// TIA Portal project "Insert_Password" (V18)

(* hardware
DEVICE "S7-1200 station_2"  S7-1200 Station
   slot 0: "Rack_0"  S7-1200 Rack  Rack  V1.0
   slot 1: "PLC_1"  CPU 1215C DC/DC/Rly  6ES7 215-1HG40-0XB0  V4.6
DEVICE "HMI_1"  KTP700 Basic PN
   slot 0: "HMI_1"  KTP700 Basic PN  6AV2 123-2GB03-0AX0  17.0.0.0
   slot 1: "HMI_RT_1"  KTP700 Basic PN  6AV2 123-2GB03-0AX0  17.0.0.0
   slot 5: "HMI_1.IE_CP_1"  PROFINET Interface  17.0.0.0
      slot 1: "PROFINET Interface_1"  PROFINET Interface
         slot 1: "Port_1"  Port
*)

// ===== PLC "PLC_1"  CPU 1215C DC/DC/Rly =====

VAR_GLOBAL   // PLC tag table "Default tag table"
   "Clock_Byte" AT %MB0 : Byte;
   "Clock_10Hz" AT %M0.0 : Bool;
   "Clock_5Hz" AT %M0.1 : Bool;
   "Clock_2.5Hz" AT %M0.2 : Bool;
   "Clock_2Hz" AT %M0.3 : Bool;
   "Clock_1.25Hz" AT %M0.4 : Bool;
   "Clock_1Hz" AT %M0.5 : Bool;
   "Clock_0.625Hz" AT %M0.6 : Bool;
   "Clock_0.5Hz" AT %M0.7 : Bool;
END_VAR

DATA_BLOCK "Logica_TIP_DB"   // DB1
{ S7_Optimized_Access := 'TRUE' }
VERSION : 0.1
// stored: InstanceOfName Logica_TIP
"Logica_TIP"
BEGIN
END_DATA_BLOCK

DATA_BLOCK "Data_block_1"   // DB3
{ S7_Optimized_Access := 'TRUE' }
VERSION : 0.1
   VAR
      Convalida_Lv1 : Bool;
      Convalida_Lv2 : Bool;
      Convalida_Lv3 : Bool;
      Disattiva : Bool;
      Selezione_modalita : Int;
      Password_1 : Array[0..15] of UInt;
      Password_2 : Array[0..15] of UInt;
      Password_3 : Array[0..15] of UInt;
      Lunghezza_Pw : Int := 8;
      richiesta_lv1 : Bool;
      richiesta_lv2 : Bool;
      richiesta_lv3 : Bool;
   END_VAR
BEGIN
   Password_1[0] := 1;
   Password_1[1] := 2;
   Password_1[2] := 1;
   Password_1[3] := 1;
   Password_2[0] := 0;
   Password_2[1] := 4;
   Password_2[2] := 0;
   Password_2[3] := 9;
   Password_3[0] := 1;
   Password_3[1] := 2;
   Password_3[2] := 3;
   Password_3[3] := 4;
   Password_1[4] := 2;
   Password_1[5] := 0;
   Password_1[6] := 2;
   Password_1[7] := 3;
   Password_2[4] := 1;
   Password_2[5] := 9;
   Password_2[6] := 9;
   Password_2[7] := 7;
   Password_3[4] := 5;
   Password_3[5] := 6;
   Password_3[6] := 7;
   Password_3[7] := 8;
   Password_3[8] := 0;
   Password_3[9] := 0;
END_DATA_BLOCK

// folder: System blocks/Program resources

DATA_BLOCK "IEC_Timer_0_DB"   // DB2
{ S7_Optimized_Access := 'TRUE' }
AUTHOR : Simatic
FAMILY : IEC
NAME : IEC_TMR
VERSION : 1.0
// stored: InstanceOfName IEC_TIMER
"IEC_TIMER"
BEGIN
END_DATA_BLOCK

DATA_BLOCK "IEC_Timer_0_DB_1"   // DB4
{ S7_Optimized_Access := 'TRUE' }
AUTHOR : Simatic
FAMILY : IEC
NAME : IEC_TMR
VERSION : 1.0
// stored: InstanceOfName IEC_TIMER
"IEC_TIMER"
BEGIN
END_DATA_BLOCK

// folder: (top level)

FUNCTION_BLOCK "Logica_TIP"   // FB2, SCL
{ S7_Optimized_Access := 'TRUE' }
VERSION : 0.1
   VAR_INPUT
      Selezione_Modalità : Int;
      Richiesta_Lv_1 : Bool;
      Richiesta_Lv_2 : Bool;
      Richiesta_Lv_3 : Bool;
      Disattiva_Abilitazioni : Bool;
   END_VAR
   VAR_OUTPUT
      Livello_1 : Bool;
      Livello_2 : Bool;
      Livello_3 : Bool;
   END_VAR
   VAR_IN_OUT
      password_1 : Array[0..#N_Array] of UInt;
      password_2 : Array[0..#N_Array] of UInt;
      password_3 : Array[0..#N_Array] of UInt;
      Lunghezza_Pw : Int;
   END_VAR
   VAR
      Array_Input : Array[0..#N_Array] of UInt;
      Array_Linee : Array[0..#N_Array] of Bool;
      Conteggio : UInt;
      Array_Memoria : Array[0..#N_Array] of Bool;
      Array_Fronti : Array[0..#N_Array] of Bool;
      Array_Fronti_Change : Array[0..#N_Array] of Bool;
      Visibilità : Bool;
      Numero : UInt;
      visibilità_Numeri : UInt;
      "Visibilità_Numeri_*" : UInt;
      "Visibilità_Numeri_°" : UInt;
      Attiva_Change : Bool;
      Stato_Cambio_Pw : UInt;
      Richiesta_Lv1 : Bool;
      Richiesta_Lv2 : Bool;
      Richiesta_Lv3 : Bool;
      Fronte_Disabilità : Bool;
      Variabili_Scritte_Change : String;
      Change_Status : UInt;
      "Password_Selected_ Change" : UInt;
      ET : Time;
      ET_1 : Time;
      appoggio_fronte_10 : Bool;
      n_div : Array[0..10] of Int;
      Scritte_Errori : String;
      vis_Scritte_Errori : Bool;
      R1 : R_TRIG;
      R2 : R_TRIG;
      R3 : R_TRIG;
      R4 : R_TRIG;
      R5 : R_TRIG;
      F_13 : F_TRIG;
      R_11 : R_TRIG;
      R_12 : R_TRIG;
      R_14 : R_TRIG;
      R_0 : R_TRIG;
      R_1 : R_TRIG;
      R_3 : R_TRIG;
      R_4 : R_TRIG;
      R_5 : R_TRIG;
      R_6 : R_TRIG;
      R_2 : R_TRIG;
      R_7 : R_TRIG;
      R_8 : R_TRIG;
      R_9 : R_TRIG;
   END_VAR
   VAR_TEMP
      n : Int;
   END_VAR
   VAR CONSTANT
      N_Array : Int := 15;
   END_VAR
BEGIN
   IF #Lunghezza_Pw > 16 THEN
       #Lunghezza_Pw := 16;
       #Scritte_Errori := 'Valore massimo inseribile: 16';
       #vis_Scritte_Errori := true;
   END_IF;

   REGION monitoro le richieste abilitazioni e attivo i vari settaggi
       #R1(CLK:=#Richiesta_Lv_1);
       #R2(CLK:=#Richiesta_Lv_2);
       #R3(CLK:=#Richiesta_Lv_3);

       IF #R1.Q THEN
           #Visibilità := true;
           #Richiesta_Lv1 := true;
       END_IF;

       IF #R2.Q THEN
           #Visibilità := true;
           #Richiesta_Lv2 := true;
       END_IF;

       IF #R3.Q THEN
           #Visibilità := true;
           #Richiesta_Lv3 := true;
       END_IF;
   END_REGION

   REGION Gestione attivazione Visibilità
       #R4(CLK := #Visibilità);
       IF #R4.Q THEN
           #Variabili_Scritte_Change := 'inserisci password';
           #visibilità_Numeri := 1;
           #Conteggio := 0;
       END_IF;
   END_REGION;

   IF #Visibilità = TRUE THEN  //verifico se la visibilità è attiva
       REGION gestione linee e numeri/asterischi
           IF "Clock_1.25Hz" = true THEN
               #Array_Linee[#Conteggio] := true;
           ELSE
               FOR #n := 0 TO #N_Array DO
                   #Array_Linee[#n] := FALSE;
               END_FOR;
           END_IF;

           #R5(CLK:="Clock_10Hz");
           IF #R5.Q THEN
               FOR #n := 0 TO #N_Array DO
                   #Array_Linee[#n] := FALSE;
               END_FOR;
           END_IF;

           #F_13(CLK:=#Array_Memoria[13]);

           IF #Array_Memoria[13] = true THEN
               #visibilità_Numeri := 2;
           END_IF;

           IF #F_13.Q THEN
               IF "IEC_Timer_0_DB_1".Q = true THEN
                   #visibilità_Numeri := 2;
               ELSE
                   #visibilità_Numeri := 1;
               END_IF;
           END_IF;


           "IEC_Timer_0_DB_1".TON(IN := #Array_Memoria[13],
                                  PT := T#1s,
                                  ET => #ET);

           CASE #visibilità_Numeri OF
               1:
                   #"Visibilità_Numeri_°" := 0;
                   #"Visibilità_Numeri_*" := #Lunghezza_Pw;
               2:
                   #"Visibilità_Numeri_°" := #Lunghezza_Pw;
                   #"Visibilità_Numeri_*" := 0;

           END_CASE;
       END_REGION

       REGION rilevamento e gestione pulsanti 
           REGION rilevamento e funzionalita pulsante esc
               // pressione pulsante "ESC"
               #R_11(CLK:=#Array_Memoria[11]);

               IF #R_11.Q THEN
                   FOR #n := 0 TO #N_Array DO
                       #Array_Input[#n] := 0;
                   END_FOR;
                   FOR #n := 0 TO #N_Array DO
                       #Array_Linee[#n] := FALSE;
                   END_FOR;
                   #Conteggio := 0;
                   #Visibilità := FALSE;
                   #Richiesta_Lv1 := false;
                   #Richiesta_Lv2 := false;
                   #Richiesta_Lv3 := false;
                   #"Visibilità_Numeri_°" := 0;
                   #"Visibilità_Numeri_*" := 0;
                   #Change_Status := 0;
               END_IF;
           END_REGION

           REGION rilevamento e funzionalità pulsante canc
               // pressione pulsante "CANC"
               #R_12(CLK:=#Array_Memoria[12]);
               IF #R_12.Q THEN
                   FOR #n := 0 TO #N_Array DO
                       #Array_Input[#n] := 0;
                   END_FOR;
                   #Conteggio := 0;
               END_IF;
           END_REGION

           REGION rilevamento e funzionalità pulsante indietro
               // pressione pulsante indietro
               #R_14(CLK:=#Array_Memoria[14]);
               IF #R_14.Q THEN
                   IF #Conteggio > 0 THEN
                       #Conteggio := #Conteggio - 1;
                       #Array_Input[#Conteggio] := 0;
                   END_IF;
               END_IF;
           END_REGION

       END_REGION

       REGION rilevazione pressione pulsanti fintanto che il numero di caratteri inseriti non superi la lunghezza_pw

           IF #Conteggio < #Lunghezza_Pw THEN  //verifico se le volte in cui i numeri sono stati premuti è minore di #lunghezza_pw

               //vado a registrare gli input dei pulsanti numerici
               #R_0(CLK:= #Array_Memoria[0]);
               #R_1(CLK:= #Array_Memoria[1]);
               #R_2(CLK:= #Array_Memoria[2]);
               #R_3(CLK:= #Array_Memoria[3]);
               #R_4(CLK := #Array_Memoria[4]);
               #R_5(CLK:= #Array_Memoria[5]);
               #R_6(CLK:= #Array_Memoria[6]);
               #R_7(CLK:= #Array_Memoria[7]);
               #R_8(CLK:= #Array_Memoria[8]);
               #R_9(CLK:= #Array_Memoria[9]);

               IF #R_0.Q THEN
                   #Array_Linee[#Numero] := FALSE;
                   #Array_Input[#Conteggio] := 0;
                   #Conteggio := #Conteggio + 1;
               END_IF;

               IF #R_1.Q THEN
                   #Array_Linee[#Numero] := FALSE;
                   #Array_Input[#Conteggio] := 1;
                   #Conteggio := #Conteggio + 1;
               END_IF;

               IF #R_2.Q  THEN
                   #Array_Linee[#Numero] := FALSE;
                   #Array_Input[#Conteggio] := 2;
                   #Conteggio := #Conteggio + 1;
               END_IF;

               IF #R_3.Q THEN
                   #Array_Linee[#Numero] := FALSE;
                   #Array_Input[#Conteggio] := 3;
                   #Conteggio := #Conteggio + 1;
               END_IF;

               IF #R_4.Q THEN
                   #Array_Linee[#Numero] := FALSE;
                   #Array_Input[#Conteggio] := 4;
                   #Conteggio := #Conteggio + 1;
               END_IF;

               IF #R_5.Q THEN
                   #Array_Linee[#Numero] := FALSE;
                   #Array_Input[#Conteggio] := 5;
                   #Conteggio := #Conteggio + 1;
               END_IF;

               IF #R_6.Q THEN
                   #Array_Linee[#Numero] := FALSE;
                   #Array_Input[#Conteggio] := 6;
                   #Conteggio := #Conteggio + 1;
               END_IF;

               IF #R_7.Q THEN
                   #Array_Linee[#Numero] := FALSE;
                   #Array_Input[#Conteggio] := 7;
                   #Conteggio := #Conteggio + 1;
               END_IF;

               IF #R_8.Q THEN
                   #Array_Linee[#Numero] := FALSE;
                   #Array_Input[#Conteggio] := 8;
                   #Conteggio := #Conteggio + 1;
               END_IF;

               IF #R_9.Q THEN
                   #Array_Linee[#Numero] := FALSE;
                   #Array_Input[#Conteggio] := 9;
                   #Conteggio := #Conteggio + 1;
               END_IF;

           END_IF;
       END_REGION

       REGION Change_Status=0
           IF #Change_Status = 0 THEN

               REGION Restituzione risultato in base alla MODalità di funzionamento selezionata

                   IF (#Array_Memoria[10] = true) & (#Array_Fronti[10] = false) THEN

                       CASE #Selezione_Modalità OF
                           0:
                               FOR #n := 0 TO (#Lunghezza_Pw - 1) DO
                                   IF #Array_Input[#n] <> #password_1[#n] THEN
                                       #n_div[0] := #n_div[0] + 1;
                                   END_IF;
                               END_FOR;
                               FOR #n := 0 TO (#Lunghezza_Pw - 1) DO
                                   IF #Array_Input[#n] <> #password_2[#n] THEN
                                       #n_div[1] := #n_div[1] + 1;
                                   END_IF;
                               END_FOR;
                               FOR #n := 0 TO (#Lunghezza_Pw - 1) DO
                                   IF #Array_Input[#n] <> #password_3[#n] THEN
                                       #n_div[2] := #n_div[2] + 1;
                                   END_IF;
                               END_FOR;
                               IF #n_div[0] = 0 THEN
                                   #Livello_1 := true;
                                   #Livello_2 := true;
                                   #Livello_3 := true;
                                   #Variabili_Scritte_Change := 'Password corretta';
                               ELSE
                                   IF #n_div[1] = 0 THEN
                                       #Livello_2 := true;
                                       #Livello_3 := true;
                                       #Variabili_Scritte_Change := 'Password corretta';
                                   ELSE
                                       IF #n_div[2] = 0 THEN
                                           #Livello_3 := true;
                                           #Variabili_Scritte_Change := 'Password corretta';
                                       ELSE
                                           #Variabili_Scritte_Change := 'Password sbagliata';
                                       END_IF;
                                   END_IF;
                               END_IF;

                                   1:
                                   IF #Richiesta_Lv1 = true THEN
                                       FOR #n := 0 TO (#Lunghezza_Pw - 1) DO
                                           IF #Array_Input[#n] <> #password_1[#n] THEN
                                               #n_div[3] := #n_div[3] + 1;
                                           END_IF;
                                       END_FOR;
                                       IF #n_div[3] = 0 THEN
                                           #Variabili_Scritte_Change := 'Password corretta';
                                           #Livello_1 := true;
                                       ELSE
                                           #Variabili_Scritte_Change := 'Password sbagliata';
                                       END_IF;
                                   END_IF;

                                   IF #Richiesta_Lv2 = true THEN
                                       FOR #n := 0 TO (#Lunghezza_Pw - 1) DO
                                           IF #Array_Input[#n] <> #password_2[#n] THEN
                                               #n_div[4] := #n_div[4] + 1;
                                           END_IF;
                                       END_FOR;
                                       IF #n_div[4] = 0 THEN
                                           #Variabili_Scritte_Change := 'Password corretta';
                                           #Livello_2 := true;
                                       ELSE
                                           #Variabili_Scritte_Change := 'Password sbagliata';
                                       END_IF;
                                   END_IF;

                                   IF #Richiesta_Lv3 = true THEN
                                       FOR #n := 0 TO (#Lunghezza_Pw - 1) DO
                                           IF #Array_Input[#n] <> #password_3[#n] THEN
                                               #n_div[5] := #n_div[5] + 1;
                                           END_IF;
                                       END_FOR;
                                       IF #n_div[5] = 0 THEN
                                           #Variabili_Scritte_Change := 'Password corretta';
                                           #Livello_3 := true;
                                       ELSE
                                           #Variabili_Scritte_Change := 'Password sbagliata';
                                       END_IF;
                                   END_IF;
                                   2:

                                   FOR #n := 0 TO (#Lunghezza_Pw - 1) DO
                                       IF #Array_Input[#n] <> #password_1[#n] THEN
                                           #n_div[6] := #n_div[6] + 1;
                                       END_IF;
                                   END_FOR;
                                   IF #n_div[6] = 0 THEN
                                       #Variabili_Scritte_Change := 'Password corretta';
                                       #Livello_1 := true;
                                       #Livello_2 := true;
                                       #Livello_3 := true;
                                   ELSE
                                       #Variabili_Scritte_Change := 'Password sbagliata';
                                   END_IF;
                       END_CASE;
                   END_IF;
                   #Array_Fronti[10] := #Array_Memoria[10];
                   #Array_Memoria[10] := false;
                   FOR #n := 0 TO 6 DO
                       #n_div[#n] := 0;
                   END_FOR;

               END_REGION

           END_IF;

       END_REGION

       REGION gestione modalità cambio password

           REGION Pressione pulsante change password ed entrata nella modalità sovrascrittura
               IF (#Array_Memoria[15] = true) & (#Array_Fronti[15] = false) THEN
                   #Variabili_Scritte_Change := 'Seleziona password';
                   FOR #n := 0 TO #N_Array DO
                       #Array_Input[#n] := 0;
                   END_FOR;
                   #Conteggio := 0;
                   #Change_Status := 1;
               END_IF;
               #Array_Fronti[15] := #Array_Memoria[15];
           END_REGION

           REGION Change_Status=1

               IF #Change_Status = 1 THEN
                   IF (#Array_Memoria[1] = true) & (#Array_Fronti_Change[1] = false) THEN
                       FOR #n := 0 TO #N_Array DO
                           #Array_Input[#n] := 0;
                       END_FOR;
                       #Conteggio := 0;
                       #Variabili_Scritte_Change := 'password precedente';
                       #Change_Status := 2;
                       #"Password_Selected_ Change" := 1;
                   END_IF;
                   #Array_Fronti_Change[1] := #Array_Memoria[1];

                   IF (#Array_Memoria[2] = true) & (#Array_Fronti_Change[2] = false) THEN
                       FOR #n := 0 TO #N_Array DO
                           #Array_Input[#n] := 0;
                       END_FOR;
                       #Conteggio := 0;
                       #Variabili_Scritte_Change := 'password precedente'; // 
                       #Change_Status := 2;
                       #"Password_Selected_ Change" := 2;
                   END_IF;
                   #Array_Fronti_Change[2] := #Array_Memoria[2];


                   IF (#Array_Memoria[3] = true) & (#Array_Fronti_Change[3] = false) THEN
                       FOR #n := 0 TO #N_Array DO
                           #Array_Input[#n] := 0;
                       END_FOR;
                       #Conteggio := 0;
                       #Variabili_Scritte_Change := 'password precedente';
                       #Change_Status := 2;
                       #"Password_Selected_ Change" := 3;
                   END_IF;
                   #Array_Fronti_Change[3] := #Array_Memoria[3];
               END_IF;

           END_REGION


           REGION Change_Status=2
               IF #Change_Status = 2 THEN
                   IF #Array_Memoria[10] = true & #Array_Fronti_Change[10] = FALSE THEN
                       CASE #"Password_Selected_ Change" OF
                           1:
                               FOR #n := 0 TO (#Lunghezza_Pw - 1) DO
                                   IF #Array_Input[#n] <> #password_1[#n] THEN
                                       #n_div[7] := #n_div[7] + 1;
                                   END_IF;
                               END_FOR;
                               IF #n_div[7] = 0  THEN
                                   #Change_Status := 3;
                                   FOR #n := 0 TO #N_Array DO
                                       #Array_Input[#n] := 0;
                                   END_FOR;
                                   #Conteggio := 0;
                                   #Variabili_Scritte_Change := 'Nuova password';
                                   GOTO end;
                               ELSE
                                   #Variabili_Scritte_Change := 'Password errata';
                               END_IF;

                           2:
                               FOR #n := 0 TO (#Lunghezza_Pw - 1) DO
                                   IF #Array_Input[#n] <> #password_2[#n] THEN
                                       #n_div[8] := #n_div[8] + 1;
                                   END_IF;
                               END_FOR;
                               IF #n_div[8] = 0 THEN
                                   #Change_Status := 3;
                                   FOR #n := 0 TO #N_Array DO
                                       #Array_Input[#n] := 0;
                                   END_FOR;
                                   #Conteggio := 0;
                                   #Variabili_Scritte_Change := 'Nuova password';
                                   GOTO end;
                               ELSE
                                   #Variabili_Scritte_Change := 'Password errata';
                               END_IF;
                           3:
                               FOR #n := 0 TO (#Lunghezza_Pw - 1) DO
                                   IF #Array_Input[#n] <> #password_3[#n] THEN
                                       #n_div[9] := #n_div[9] + 1;
                                   END_IF;
                               END_FOR;
                               IF #n_div[9] = 0 THEN
                                   #Change_Status := 3;
                                   FOR #n := 0 TO #N_Array DO
                                       #Array_Input[#n] := 0;
                                   END_FOR;
                                   #Conteggio := 0;
                                   #Variabili_Scritte_Change := 'Nuova password';
                                   GOTO end;
                               ELSE
                                   #Variabili_Scritte_Change := 'Password errata';
                               END_IF;
                       END_CASE;
                   END_IF;
                   #Array_Fronti_Change[10] := #Array_Memoria[10];
               END_IF;


           END_REGION


           REGION Change_Status=3
               IF #Change_Status = 3 THEN
                   IF #Array_Memoria[10] = true & #Array_Fronti_Change[11] = FALSE THEN
                       #appoggio_fronte_10 := true;
                       #Variabili_Scritte_Change := 'Password modificata';
                   END_IF;
                   "IEC_Timer_0_DB".TON(IN := #appoggio_fronte_10,
                                        PT := T#1s,
                                        ET => #ET_1);
                   IF "IEC_Timer_0_DB".Q = true THEN
                       #appoggio_fronte_10 := false;
                       CASE #"Password_Selected_ Change" OF
                           1:
                               #"password_1" := #Array_Input;
                               GOTO esc;
                           2:
                               #"password_2" := #Array_Input;
                               GOTO esc;
                           3:
                               #"password_3" := #Array_Input;
                               GOTO esc;
                       END_CASE;
                   esc:
                       FOR #n := 0 TO #N_Array DO
                           #Array_Input[#n] := 0;
                       END_FOR;
                       FOR #n := 0 TO #N_Array DO
                           #Array_Linee[#n] := FALSE;
                       END_FOR;
                       #Conteggio := 0;
                       #Visibilità := FALSE;
                       #Richiesta_Lv1 := false;
                       #Richiesta_Lv2 := false;
                       #Richiesta_Lv3 := false;
                       #"Visibilità_Numeri_°" := 0;
                       #"Visibilità_Numeri_*" := 0;
                       #Change_Status := 0;
                   END_IF;
                   #Array_Fronti_Change[11] := #Array_Memoria[10];
                   #Array_Memoria[10] := false;
               END_IF;


           END_REGION

       end:
           #Array_Memoria[10] := false;
           FOR #n := 7 TO 9 DO
               #n_div[#n] := 0;
           END_FOR;
       END_REGION


   END_IF;

   REGION rilevamento e funzionalità pulsante disattiva abilitazioni
       // va fuori dal controllo visibilità altrimenti non funziona
       IF #Disattiva_Abilitazioni = true & #Fronte_Disabilità = false THEN
           #Livello_1 := false;
           #Livello_2 := false;
           #Livello_3 := false;
       END_IF;
       #Fronte_Disabilità := #Disattiva_Abilitazioni;
   END_REGION
END_FUNCTION_BLOCK

ORGANIZATION_BLOCK "Main"   // OB1, LAD, ProgramCycle
TITLE = "Main Program Sweep (Cycle)"
{ S7_Optimized_Access := 'TRUE' }
VERSION : 0.1
   VAR_INPUT
      Initial_Call : Bool;   // Initial call of this OB
      Remanence : Bool;   // =True, if remanent data are available
   END_VAR
BEGIN

REGION Network 1
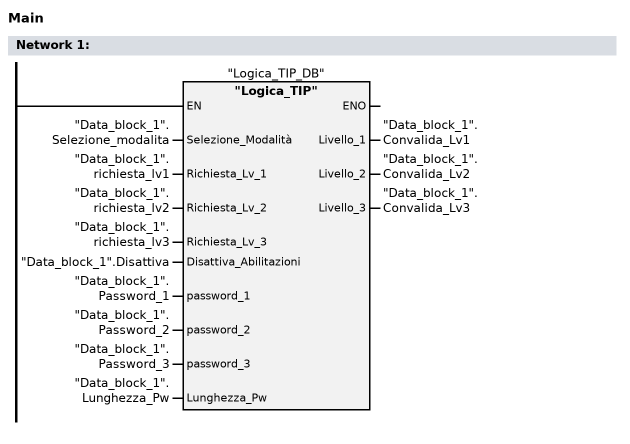
   RUNG wire#powerrail
      "Logica_TIP_DB"(Selezione_Modalità := "Data_block_1".Selezione_modalita, Richiesta_Lv_1 := "Data_block_1".richiesta_lv1, Richiesta_Lv_2 := "Data_block_1".richiesta_lv2, Richiesta_Lv_3 := "Data_block_1".richiesta_lv3, Disattiva_Abilitazioni := "Data_block_1".Disattiva, Lunghezza_Pw := "Data_block_1".Lunghezza_Pw, password_1 := "Data_block_1".Password_1, password_2 := "Data_block_1".Password_2, password_3 := "Data_block_1".Password_3, Livello_1 => "Data_block_1".Convalida_Lv1, Livello_2 => "Data_block_1".Convalida_Lv2, Livello_3 => "Data_block_1".Convalida_Lv3)
   END_RUNG
   // the same network as SCL:
   "Logica_TIP_DB"(Selezione_Modalità := "Data_block_1".Selezione_modalita,   // "Logica_TIP"
                   Richiesta_Lv_1 := "Data_block_1".richiesta_lv1,
                   Richiesta_Lv_2 := "Data_block_1".richiesta_lv2,
                   Richiesta_Lv_3 := "Data_block_1".richiesta_lv3,
                   Disattiva_Abilitazioni := "Data_block_1".Disattiva,
                   password_1 := "Data_block_1".Password_1,
                   password_2 := "Data_block_1".Password_2,
                   password_3 := "Data_block_1".Password_3,
                   Lunghezza_Pw := "Data_block_1".Lunghezza_Pw,
                   Livello_1 => "Data_block_1".Convalida_Lv1,
                   Livello_2 => "Data_block_1".Convalida_Lv2,
                   Livello_3 => "Data_block_1".Convalida_Lv3);
END_REGION
END_ORGANIZATION_BLOCK

(* ===== HMI "HMI_RT_1" =====
system functions are stored by id; their names below are inferred from use
connection "HMI_Connection_1": ETHERNET, SMART_S7_1200_OMS

HMI tags "Default tag table"
   "Tag_ScreenNumber" : UInt, internal
   "Variabili_Visibilità" : Bool = PLC Logica_TIP_DB.Visibilità, 100 ms
   "Variabili_Array_Memoria{12}" : Bool = PLC Logica_TIP_DB.Array_Memoria[12], 100 ms
   "Variabili_Array_Memoria{10}" : Bool = PLC Logica_TIP_DB.Array_Memoria[10], 100 ms
   "Variabili_Array_Memoria{11}" : Bool = PLC Logica_TIP_DB.Array_Memoria[11], 100 ms
   "Variabili_Array_Memoria{0}" : Bool = PLC Logica_TIP_DB.Array_Memoria[0], 100 ms
   "Variabili_Array_Memoria{9}" : Bool = PLC Logica_TIP_DB.Array_Memoria[9], 100 ms
   "Variabili_Array_Memoria{8}" : Bool = PLC Logica_TIP_DB.Array_Memoria[8], 100 ms
   "Variabili_Array_Memoria{1}" : Bool = PLC Logica_TIP_DB.Array_Memoria[1], 100 ms
   "Variabili_Array_Memoria{2}" : Bool = PLC Logica_TIP_DB.Array_Memoria[2], 100 ms
   "Variabili_Array_Memoria{3}" : Bool = PLC Logica_TIP_DB.Array_Memoria[3], 100 ms
   "Variabili_Array_Memoria{4}" : Bool = PLC Logica_TIP_DB.Array_Memoria[4], 100 ms
   "Variabili_Array_Memoria{5}" : Bool = PLC Logica_TIP_DB.Array_Memoria[5], 100 ms
   "Variabili_Array_Memoria{6}" : Bool = PLC Logica_TIP_DB.Array_Memoria[6], 100 ms
   "Variabili_Array_Memoria{7}" : Bool = PLC Logica_TIP_DB.Array_Memoria[7], 100 ms
   "Variabili_Array_Input{0}" : UInt = PLC Logica_TIP_DB.Array_Input[0], 100 ms
   "Variabili_Array_Input{2}" : UInt = PLC Logica_TIP_DB.Array_Input[2], 100 ms
   "Variabili_Array_Input{1}" : UInt = PLC Logica_TIP_DB.Array_Input[1], 100 ms
   "Variabili_Array_Input{3}" : UInt = PLC Logica_TIP_DB.Array_Input[3], 100 ms
   "Variabili_Array_Memoria{13}" : Bool = PLC Logica_TIP_DB.Array_Memoria[13], 100 ms
   "Variabili_visibilità_Numeri" : UInt = PLC Logica_TIP_DB.visibilità_Numeri, 100 ms
   "Variabili_Array_Memoria{14}" : Bool = PLC Logica_TIP_DB.Array_Memoria[14], 100 ms
   "Data_block_1_Disattiva" : Bool = PLC Data_block_1.Disattiva, 100 ms
   "Data_block_1_Richiesta_Lv1" : Bool = PLC Data_block_1.richiesta_lv1, 100 ms
   "Data_block_1_RIchiesta_Lv2" : Bool = PLC Data_block_1.richiesta_lv2, 100 ms
   "Data_block_1_Richiesta_Lv3" : Bool = PLC Data_block_1.richiesta_lv3, 100 ms
   "Data_block_1_Disattiva(1)" : Bool = PLC Data_block_1.Disattiva, 100 ms
   "Variabili_Visibilità_Numeri_*" : UInt = PLC Logica_TIP_DB.Visibilità_Numeri_*, 100 ms
   "Variabili_Visibilità_Numeri_°" : UInt = PLC Logica_TIP_DB.Visibilità_Numeri_°, 100 ms
   "Variabili_Array_Input{4}" : UInt = PLC Logica_TIP_DB.Array_Input[4], 100 ms
   "Variabili_Array_Input{5}" : UInt = PLC Logica_TIP_DB.Array_Input[5], 100 ms
   "Variabili_Array_Input{6}" : UInt = PLC Logica_TIP_DB.Array_Input[6], 100 ms
   "Variabili_Array_Input{7}" : UInt = PLC Logica_TIP_DB.Array_Input[7], 100 ms
   "Variabili_Array_Input{8}" : UInt = PLC Logica_TIP_DB.Array_Input[8], 100 ms
   "Variabili_Array_Input{9}" : UInt = PLC Logica_TIP_DB.Array_Input[9], 100 ms
   "Variabili_Array_Input{10}" : UInt = PLC Logica_TIP_DB.Array_Input[10], 100 ms
   "Variabili_Array_Input{11}" : UInt = PLC Logica_TIP_DB.Array_Input[11], 100 ms
   "Variabili_Array_Linee{0}" : Bool = PLC Logica_TIP_DB.Array_Linee[0], 100 ms
   "Variabili_Array_Linee{1}" : Bool = PLC Logica_TIP_DB.Array_Linee[1], 100 ms
   "Variabili_Array_Linee{2}" : Bool = PLC Logica_TIP_DB.Array_Linee[2], 100 ms
   "Variabili_Array_Linee{3}" : Bool = PLC Logica_TIP_DB.Array_Linee[3], 100 ms
   "Variabili_Array_Linee{4}" : Bool = PLC Logica_TIP_DB.Array_Linee[4], 100 ms
   "Variabili_Array_Linee{5}" : Bool = PLC Logica_TIP_DB.Array_Linee[5], 100 ms
   "Variabili_Array_Linee{6}" : Bool = PLC Logica_TIP_DB.Array_Linee[6], 100 ms
   "Variabili_Array_Linee{7}" : Bool = PLC Logica_TIP_DB.Array_Linee[7], 100 ms
   "Variabili_Array_Linee{8}" : Bool = PLC Logica_TIP_DB.Array_Linee[8], 100 ms
   "Variabili_Array_Linee{9}" : Bool = PLC Logica_TIP_DB.Array_Linee[9], 100 ms
   "Variabili_Array_Linee{10}" : Bool = PLC Logica_TIP_DB.Array_Linee[10], 100 ms
   "Variabili_Array_Linee{11}" : Bool = PLC Logica_TIP_DB.Array_Linee[11], 100 ms
   "Variabili_Array_Linee{12}" : Bool = PLC Logica_TIP_DB.Array_Linee[12], 100 ms
   "Variabili_Array_Memoria{15}" : Bool = PLC Logica_TIP_DB.Array_Memoria[15], 100 ms
   "Logica_PW_DB_Variabili_Scritte_Change" : String[254] = PLC Logica_TIP_DB.Variabili_Scritte_Change, 100 ms
   "Logica_PW_DB_Change_Status" : UInt = PLC Logica_TIP_DB.Change_Status AT %DB1.DBW0, 100 ms
   "Data_block_1_Convalida_Lv1" : Bool = PLC Data_block_1.Convalida_Lv1, 100 ms
   "Data_block_1_Convalida_Lv2" : Bool = PLC Data_block_1.Convalida_Lv2, 100 ms
   "Data_block_1_Convalida_Lv3" : Bool = PLC Data_block_1.Convalida_Lv3, 100 ms
   "Data_block_1_Selezione_modalita" : Int = PLC Data_block_1.Selezione_modalita, 100 ms
   "Data_block_1_Lunghezza_Pw" : Int = PLC Data_block_1.Lunghezza_Pw, 100 ms
   "Logica_TIP_DB_Scritte_Errori" : String[254] = PLC Logica_TIP_DB.Scritte_Errori, 1 s
   "Logica_TIP_DB_vis_Scritte_Errori" : Bool = PLC Logica_TIP_DB.vis_Scritte_Errori, 1 s

screen "Screen_1" 800x480
   Button "Button_14" at 659,33 size 96x32; TextOff 'PW1'
      on Press: function_b14e0dd5("Data_block_1_Richiesta_Lv1", 0)
      Visibility <- "Variabili_Visibilità"
   Button "Button_17" at 659,200 size 96x32; TextOff 'Disatt.'
      on Press: function_b14e0dd5("Data_block_1_Disattiva", 0)
      Visibility <- "Variabili_Visibilità"
   Button "Button_16" at 659,84 size 96x32; TextOff 'PW2'
      on Press: function_b14e0dd5("Data_block_1_RIchiesta_Lv2", 0)
      Visibility <- "Variabili_Visibilità"
   Button "Button_18" at 659,142 size 96x32; TextOff 'PW3'
      on Press: function_b14e0dd5("Data_block_1_Richiesta_Lv3", 0)
      Visibility <- "Variabili_Visibilità"
   Rectangle "Rectangle_2" at 22,17 size 220x324
      Visibility <- "Variabili_Visibilità"
   Button "Button_1" at 27,229 size 65x50; TextOff '1'
      on Press: function_b14e0dd5("Variabili_Array_Memoria{1}", 0)
      Visibility <- "Variabili_Visibilità"
   Button "Button_2" at 100,229 size 65x50; TextOff '2'
      on Press: function_b14e0dd5("Variabili_Array_Memoria{2}", 0)
      Visibility <- "Variabili_Visibilità"
   Button "Button_3" at 172,229 size 65x50; TextOff '3'
      on Press: function_b14e0dd5("Variabili_Array_Memoria{3}", 0)
      Visibility <- "Variabili_Visibilità"
   Button "Button_4" at 27,173 size 65x50; TextOff '4'
      on Press: function_b14e0dd5("Variabili_Array_Memoria{4}", 0)
      Visibility <- "Variabili_Visibilità"
   Button "Button_5" at 100,173 size 65x50; TextOff '5'
      on Press: function_b14e0dd5("Variabili_Array_Memoria{5}", 0)
      Visibility <- "Variabili_Visibilità"
   Button "Button_6" at 172,173 size 65x50; TextOff '6'
      on Press: function_b14e0dd5("Variabili_Array_Memoria{6}", 0)
      Visibility <- "Variabili_Visibilità"
   Button "Button_7" at 27,118 size 65x50; TextOff '7'
      on Press: function_b14e0dd5("Variabili_Array_Memoria{7}", 0)
      Visibility <- "Variabili_Visibilità"
   Button "Button_8" at 100,118 size 65x50; TextOff '8'
      on Press: function_b14e0dd5("Variabili_Array_Memoria{8}", 0)
      Visibility <- "Variabili_Visibilità"
   Button "Button_9" at 172,118 size 65x50; TextOff '9'
      on Press: function_b14e0dd5("Variabili_Array_Memoria{9}", 0)
      Visibility <- "Variabili_Visibilità"
   Button "Button_10" at 27,285 size 65x50; TextOff '0'
      on Press: function_b14e0dd5("Variabili_Array_Memoria{0}", 0)
      Visibility <- "Variabili_Visibilità"
   Rectangle "Rectangle_3" at 22,17 size 220x32
      Visibility <- "Variabili_Visibilità"
   Button "Button_11" at 207,17 size 35x32; TextOff 'X'
      on Press: function_b14e0dd5("Variabili_Array_Memoria{11}", 0)
      Visibility <- "Variabili_Visibilità"
   Rectangle "Rectangle_1" at 25,54 size 214x60
      Visibility <- "Variabili_Visibilità"
      Appearance <- "Logica_PW_DB_Change_Status"
   Button "Button_13" at 209,87 size 28x25; TextOff 'X'
      on Press: function_b14e0dd5("Variabili_Array_Memoria{12}", 0)
      Visibility <- "Variabili_Visibilità"
   Button "Button_15" at 205,54 size 34x31; TextOff 'vis'; PictureOff "simbolo-di-vettore-dell-icona-occhio-stile-piano-progettazione-illustrazione"
      on Press: function_b14e0dd5("Variabili_Array_Memoria{13}", 0)
      Visibility <- "Variabili_Visibilità"
   Line "Line_1" at 25,84 size 214x0
      Visibility <- "Variabili_Visibilità"
   Group "Group" at 24,78 size 174x44
   Group "Group_1" at 24,87 size 174x32
   Line "Line_2" at 28,93 size 0x15
      Visibility <- "Variabili_Array_Linee{0}"
   Line "Line_3" at 41,93 size 0x15
      Visibility <- "Variabili_Array_Linee{1}"
   Line "Line_4" at 55,93 size 0x15
      Visibility <- "Variabili_Array_Linee{2}"
   Line "Line_5" at 69,93 size 0x15
      Visibility <- "Variabili_Array_Linee{3}"
   Line "Line_6" at 83,93 size 0x15
      Visibility <- "Variabili_Array_Linee{4}"
   Line "Line_7" at 97,93 size 0x15
      Visibility <- "Variabili_Array_Linee{5}"
   Line "Line_8" at 111,93 size 0x15
      Visibility <- "Variabili_Array_Linee{6}"
   Line "Line_9" at 125,93 size 0x15
      Visibility <- "Variabili_Array_Linee{7}"
   Line "Line_10" at 138,93 size 0x15
      Visibility <- "Variabili_Array_Linee{8}"
   Line "Line_11" at 152,93 size 0x15
      Visibility <- "Variabili_Array_Linee{9}"
   Line "Line_12" at 167,93 size 0x15
      Visibility <- "Variabili_Array_Linee{10}"
   Line "Line_13" at 181,93 size 0x15
      Visibility <- "Variabili_Array_Linee{11}"
   Line "Line_14" at 196,93 size 0x15
      Visibility <- "Variabili_Array_Linee{12}"
   Button "Button_19" at 172,285 size 65x50; TextOff 'ok'
      on Click: SetBit("Variabili_Array_Memoria{10}")
      Visibility <- "Variabili_Visibilità"
   Button "Button_12" at 100,285 size 65x50; TextOff '<--'; PictureOff "freccia"
      on Press: function_b14e0dd5("Variabili_Array_Memoria{14}", 0)
      Visibility <- "Variabili_Visibilità"
   Button "Button_20" at 261,28 size 65x50; TextOff 'change'
      on Press: function_b14e0dd5("Variabili_Array_Memoria{15}", 0)
      Visibility <- "Variabili_Visibilità"
   IOField "I/O field_13" at 25,55 size 185x32; FormatPattern ????????????????????????????????????????????????????????????????????????????????
      Visibility <- "Variabili_Visibilità"
      ProcessValue <- "Logica_PW_DB_Variabili_Scritte_Change"
   GraphicIOField "PlotLight_Round_G" at 593,24 size 50x50; PictureOff "PilotLight_Round_G_Off_256c"; PictureOn "PilotLight_Round_G_On_256c"
      ProcessValue <- "Data_block_1_Convalida_Lv1"
   GraphicIOField "PlotLight_Round_GN" at 593,75 size 50x50; PictureOff "PilotLight_Round_GN_Off_256c"; PictureOn "PilotLight_Round_GN_On_256c"
      ProcessValue <- "Data_block_1_Convalida_Lv2"
   GraphicIOField "PlotLight_Round_N_Mono" at 593,133 size 50x50; PictureOff "PilotLight_Round_N_Off_mono"; PictureOn "PilotLight_Round_N_On_mono"
      ProcessValue <- "Data_block_1_Convalida_Lv3"
   IOField "I/O field_14" at 659,247 size 96x32; FormatPattern s99999
      ProcessValue <- "Data_block_1_Selezione_modalita"
   IOField "I/O field_15" at 659,297 size 96x32; FormatPattern s99999
      ProcessValue <- "Data_block_1_Lunghezza_Pw"
   TextField "Text field_1" at 286,252 size 353x23; Text 'Selezione della modalita di funzionamento'
   TextField "Text field_2" at 330,302 size 309x23; Text 'Selezione numero caratteri password'
   Group "Group_2" at 413,341 size 374x77
   IOField "I/O field_9" at 135,78 size 21x44; FormatPattern 9
      ProcessValue <- "Variabili_Array_Input{8}"
      Visibility <- "Variabili_Visibilità_Numeri_°"
   IOField "I/O field_10" at 148,78 size 21x44; FormatPattern 9
      ProcessValue <- "Variabili_Array_Input{9}"
      Visibility <- "Variabili_Visibilità_Numeri_°"
   IOField "I/O field_11" at 163,78 size 21x44; FormatPattern 9
      ProcessValue <- "Variabili_Array_Input{10}"
      Visibility <- "Variabili_Visibilità_Numeri_°"
   IOField "I/O field_12" at 177,78 size 21x44; FormatPattern 9
      ProcessValue <- "Variabili_Array_Input{11}"
      Visibility <- "Variabili_Visibilità_Numeri_°"
   IOField "I/O field_1" at 24,78 size 21x44; FormatPattern 9
      Visibility <- "Variabili_Visibilità_Numeri_°"
      ProcessValue <- "Variabili_Array_Input{0}"
   IOField "I/O field_2" at 37,78 size 21x44; FormatPattern 9
      Visibility <- "Variabili_Visibilità_Numeri_°"
      ProcessValue <- "Variabili_Array_Input{1}"
   IOField "I/O field_3" at 52,78 size 21x44; FormatPattern 9
      Visibility <- "Variabili_Visibilità_Numeri_°"
      ProcessValue <- "Variabili_Array_Input{2}"
   IOField "I/O field_4" at 65,78 size 21x44; FormatPattern 9
      Visibility <- "Variabili_Visibilità_Numeri_°"
      ProcessValue <- "Variabili_Array_Input{3}"
   IOField "I/O field_5" at 79,78 size 21x44; FormatPattern 9
      ProcessValue <- "Variabili_Array_Input{4}"
      Visibility <- "Variabili_Visibilità_Numeri_°"
   IOField "I/O field_6" at 93,78 size 21x44; FormatPattern 9
      ProcessValue <- "Variabili_Array_Input{5}"
      Visibility <- "Variabili_Visibilità_Numeri_°"
   IOField "I/O field_7" at 107,78 size 21x44; FormatPattern 9
      ProcessValue <- "Variabili_Array_Input{6}"
      Visibility <- "Variabili_Visibilità_Numeri_°"
   IOField "I/O field_8" at 121,78 size 21x44; FormatPattern 9
      ProcessValue <- "Variabili_Array_Input{7}"
      Visibility <- "Variabili_Visibilità_Numeri_°"
   TextField "Text field_16" at 135,87 size 20x32; Text '*'
      Visibility <- "Variabili_Visibilità_Numeri_*"
   TextField "Text field_17" at 163,87 size 20x32; Text '*'
      Visibility <- "Variabili_Visibilità_Numeri_*"
   TextField "Text field_18" at 149,87 size 20x32; Text '*'
      Visibility <- "Variabili_Visibilità_Numeri_*"
   TextField "Text field_19" at 178,87 size 20x32; Text '*'
      Visibility <- "Variabili_Visibilità_Numeri_*"
   TextField "Text field_8" at 80,87 size 20x32; Text '*'
      Visibility <- "Variabili_Visibilità_Numeri_*"
   TextField "Text field_9" at 108,87 size 20x32; Text '*'
      Visibility <- "Variabili_Visibilità_Numeri_*"
   TextField "Text field_10" at 93,87 size 20x32; Text '*'
      Visibility <- "Variabili_Visibilità_Numeri_*"
   TextField "Text field_11" at 121,87 size 20x32; Text '*'
      Visibility <- "Variabili_Visibilità_Numeri_*"
   TextField "Text field_4" at 24,87 size 20x32; Text '*'
      Visibility <- "Variabili_Visibilità_Numeri_*"
   TextField "Text field_5" at 52,87 size 20x32; Text '*'
      Visibility <- "Variabili_Visibilità_Numeri_*"
   TextField "Text field_6" at 38,87 size 20x32; Text '*'
      Visibility <- "Variabili_Visibilità_Numeri_*"
   TextField "Text field_7" at 65,87 size 20x32; Text '*'
      Visibility <- "Variabili_Visibilità_Numeri_*"
   IOField "I/O field_16" at 413,341 size 374x77; FormatPattern ??????????????????????????????
      Visibility <- "Logica_TIP_DB_vis_Scritte_Errori"
      ProcessValue <- "Logica_TIP_DB_Scritte_Errori"
   Button "Button_21" at 726,354 size 50x50; TextOff 'OK'
      on Click: ResetBit("Logica_TIP_DB_vis_Scritte_Errori")
      Visibility <- "Logica_TIP_DB_vis_Scritte_Errori"

Template "Template_1" 800x480
   Button "Exit" at 714,429 size 71x50; TextOn 'Exit'; TextOff 'Exit'; PictureOn "ExitRuntime_KTP700_Basic_PN_TR"; PictureOff "ExitRuntime_KTP700_Basic_PN_TR"
      on Release: StopRuntime(0)
   Button "Template_Button" at 614,429 size 71x50; TextOff 'Text'
   Button "Template_Button_1" at 514,429 size 71x50; TextOff 'Text'
   Button "Template_Button_2" at 414,429 size 71x50; TextOff 'Text'
   Button "Template_Button_3" at 314,429 size 71x50; TextOff 'Text'
   Button "Template_Button_4" at 214,429 size 71x50; TextOff 'Text'
   Button "Alarms" at 114,429 size 71x50; TextOn 'Alarms'; TextOff 'Alarms'; PictureOn "AlarmDisplay_KTP700_Basic_PN_TR"; PictureOff "AlarmDisplay_KTP700_Basic_PN_TR"
      on Release: function_ef3f5d25("Alarm window_Unacknowledged", -1)
   Button "Start screen" at 14,429 size 71x50; TextOn 'Start screen'; TextOff 'Start screen'; PictureOn "NavigateHome_KTP700_Basic_PN_TR"; PictureOff "NavigateHome_KTP700_Basic_PN_TR"
      on Release: ActivateScreen("Screen_1", 0)
   SymbolicIOField "Symbolic_IO_Field_Screen" at 93,9 size 600x33; TextOn '1'; TextOff '0'; TextList "TextList_ScreenNames"
      on Change: ActivateScreenByNumber("Tag_ScreenNumber", 0)
      ProcessValue <- "Tag_ScreenNumber"
   DateTimeField "HmiScreenItemData" at 695,25 size 105x25
   DateTimeField "HmiScreenItemData_1" at 695,0 size 105x25
   GraphicView "Logo" at 0,0 size 91x51; Picture "Logo of HMI_1"
*)